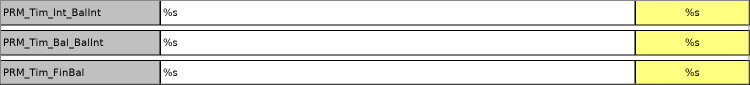
VISUALIZATION VISU_CONFIG_INTERJOINT  // 750x85
(*visualistion pour secondaire dans chambre et primaire dans sas ==> paramètres pour chambre*)
VAR_IN_OUT
	m_Input_Pompage : BLOCK_POMP_1E_PCR_PPM_ASS_ETHERCAT_SINGER;
END_VAR
    Rectangle (160,0 475x25), "%s", text list: 'TextList_Config_Pompage', text index: 17
    Rectangle (635,0 115x25), "%s", text variable: m_Input_Pompage.PRM_Tim_Int_BalInt, input disabled if: NOT Global_Variables.PRG_USER.ACTU_USER.CONF_MACHINE
        OnMouseClick: write the text variable via InputWithLimits
    Rectangle (0,0 160x25), "PRM_Tim_Int_BalInt"
    Rectangle (160,30 475x25), "%s", text list: 'TextList_Config_Pompage', text index: 18
    Rectangle (635,30 115x25), "%s", text variable: m_Input_Pompage.PRM_Tim_Bal_BalInt, input disabled if: NOT Global_Variables.PRG_USER.ACTU_USER.CONF_MACHINE
        OnMouseClick: write the text variable via InputWithLimits
    Rectangle (0,30 160x25), "PRM_Tim_Bal_BalInt"
    Rectangle (0,60 160x25), "PRM_Tim_FinBal"
    Rectangle (160,60 475x25), "%s", text list: 'TextList_Config_Pompage', text index: 19
    Rectangle (635,60 115x25), "%s", text variable: m_Input_Pompage.PRM_Tim_FinBal, input disabled if: NOT Global_Variables.PRG_USER.ACTU_USER.CONF_MACHINE
        OnMouseClick: write the text variable via InputWithLimits
END_VISUALIZATION

(* stored: Version 1.1.0.1, ProductVersion 3.1.4024.12
   Visu VISU_CONFIG_INTERJOINT: Id {692489ca-d39f-414e-b401-071f1eb13770} *)
